// TIA Portal V18 export
FUNCTION "mot_inertia_speed" : Void   // FC27, FBD
{ S7_Optimized_Access := 'TRUE' }
VERSION : 0.1
// stored: AutoNumber true, IsIECCheckEnabled false, SetENOAutomatically false, UDAEnableTagReadback false
   VAR_INPUT
      set_speed : Real;
      par : "typeMotPara";
      seconds_per_clock : Real;
   END_VAR
   VAR_OUTPUT
      ER_SET : Bool;
   END_VAR
   VAR_IN_OUT
      speed : Real;
   END_VAR
   VAR_TEMP
      v_delta : Real;
      v_step_per_cycle_max : Real;
      abs_max_speed : Real;
      time_abs_max : Real;
   END_VAR
BEGIN

REGION Network 2 (SCL)
   #v_delta := ABS(#speed - #set_speed);
   #abs_max_speed := #par.v_absoluteMax_LOGIC;
   #time_abs_max := #par.t_acc_50Hz_USER;
   #ER_SET := #abs_max_speed <= 0 OR #time_abs_max <= 0 OR #seconds_per_clock <= 0;

   #v_step_per_cycle_max := #abs_max_speed / #time_abs_max * #seconds_per_clock;
   IF #ER_SET THEN
       #speed := 0;
   ELSE
       IF #v_delta < #v_step_per_cycle_max THEN
           #speed := #set_speed;
       ELSE
           IF #set_speed > #speed THEN
               #speed := #speed + #v_step_per_cycle_max;
           ELSE
               #speed := #speed - #v_step_per_cycle_max;
           END_IF;
       END_IF;
   END_IF;
END_REGION
END_FUNCTION
